        rq_set_pos_spd_for(128, 127, 127, "1")
        rq_wait_pos_spe_for_request(128, 127, 127, "1")
        rq_go_to("1")
        rq_wait("1")
        # end: URCap Program Node
        $ 793 "cur_pose≔pose_trans(pose_inv(stn5_plane), get_actual_tcp_pose())"
        global cur_pose= pose_trans ( pose_inv (stn5_plane),  get_actual_tcp_pose ())
        $ 795 "stn5_cw_pick_p≔pose_trans(cur_pose, p[0,0,stn5_pick_cw_z/1000,0,0,0])"
        global stn5_cw_pick_p= pose_trans (cur_pose, p[0,0,stn5_pick_cw_z/1000,0,0,0])
        $ 796 "FahreLinear"
        $ 797 "stn5_cw_pick_p" "breakAfter"
        set_tcp(p[-3.0E-4,2.5E-4,0.1575,0.0,0.0,0.0])
        movel(pose_trans(stn5_plane, stn5_cw_pick_p), a=0.3, v=0.1)
        # begin: URCap Program Node
        #   Source: Robotiq_Grippers, 1.8.13.22852, Robotiq Inc.
        #   Type: Greifer
        $ 798 "Greifer geschlossen (1)"
        if not(gripper_connected[0]):
          popup("Greifer 1 muss verbunden sein, um dieses Programm auszuführen.", "Keine Verbindung", False, True, True)
        end
        if not(rq_is_gripper_activated("1")):
          popup("Greifer 1 ist nicht aktiviert. Wechseln Sie zur Registerkarte Installation > Greifer, um ihn zu aktivieren und das Programm erneut auszuführen.", "Nicht aktiviert", False, True, True)
        end
        rq_set_pos_spd_for(255, 128, 128, "1")
        rq_wait_pos_spe_for_request(255, 128, 128, "1")
        rq_go_to("1")
        rq_wait("1")
        # end: URCap Program Node
        $ 799 "source_p" "breakAfter"
        set_tcp(p[-3.0E-4,2.5E-4,0.1575,0.0,0.0,0.0])
        movel(pose_trans(stn5_plane, source_p), a=0.3, v=0.1)
        $ 800 "FahreAchse"
        $ 801 "dest_p" "breakAfter"
        set_tcp(p[-3.0E-4,2.5E-4,0.1575,0.0,0.0,0.0])
        movej(pose_trans(stn5_plane, dest_p), a=1.3962634015954636, v=1.0471975511965976)
        $ 802 "cur_pose≔pose_trans(pose_inv(stn5_plane), get_actual_tcp_pose())"
        global cur_pose= pose_trans ( pose_inv (stn5_plane),  get_actual_tcp_pose ())
        $ 804 "stn5_cw_place_p≔pose_trans(cur_pose, p[0,0,stn5_place_tb_z/1000,0,0,0])"
        global stn5_cw_place_p= pose_trans (cur_pose, p[0,0,stn5_place_tb_z/1000,0,0,0])
        $ 805 "FahreLinear"
        $ 806 "stn5_cw_place_p" "breakAfter"
        set_tcp(p[-3.0E-4,2.5E-4,0.1575,0.0,0.0,0.0])
        movel(pose_trans(stn5_plane, stn5_cw_place_p), a=0.3, v=0.1)
        # begin: URCap Program Node
        #   Source: Robotiq_Grippers, 1.8.13.22852, Robotiq Inc.
        #   Type: Greifer
        $ 807 "Greiferbewegung50% (1)"
        if not(gripper_connected[0]):
          popup("Greifer 1 muss verbunden sein, um dieses Programm auszuführen.", "Keine Verbindung", False, True, True)
        end
        if not(rq_is_gripper_activated("1")):
          popup("Greifer 1 ist nicht aktiviert. Wechseln Sie zur Registerkarte Installation > Greifer, um ihn zu aktivieren und das Programm erneut auszuführen.", "Nicht aktiviert", False, True, True)
        end
        rq_set_pos_spd_for(127, 127, 127, "1")
        rq_wait_pos_spe_for_request(127, 127, 127, "1")
        rq_go_to("1")
        rq_wait("1")
        # end: URCap Program Node
        $ 808 "dest_p" "breakAfter"
        set_tcp(p[-3.0E-4,2.5E-4,0.1575,0.0,0.0,0.0])
        movel(pose_trans(stn5_plane, dest_p), a=0.3, v=0.1)
        # begin: URCap Program Node
        #   Source: Robotiq_Grippers, 1.8.13.22852, Robotiq Inc.
        #   Type: Greifer
        $ 809 "Greifer geschlossen (1)"
        if not(gripper_connected[0]):
          popup("Greifer 1 muss verbunden sein, um dieses Programm auszuführen.", "Keine Verbindung", False, True, True)
        end
        if not(rq_is_gripper_activated("1")):
          popup("Greifer 1 ist nicht aktiviert. Wechseln Sie zur Registerkarte Installation > Greifer, um ihn zu aktivieren und das Programm erneut auszuführen.", "Nicht aktiviert", False, True, True)
        end
        rq_set_pos_spd_for(255, 255, 0, "1")
        rq_wait_pos_spe_for_request(255, 255, 0, "1")
        rq_go_to("1")
        rq_wait("1")
        # end: URCap Program Node
        $ 810 "FahreAchse"
        $ 811 "stn5_stn4_hlp_p" "breakAfter"
        set_tcp(p[-3.0E-4,2.5E-4,0.1575,0.0,0.0,0.0])
        movej(get_inverse_kin(pose_trans(stn6_plane, pose_trans(p[.776557109756, -.878329076792, .250244777977, -.001605684562, .009314448336, 1.565629725105], stn5_stn4_hlp_p_p)), qnear=stn5_stn4_hlp_p_q), a=1.3962634015954636, v=1.0471975511965976)
        $ 812 "stn6_home_p" "breakAfter"
        set_tcp(p[-3.0E-4,2.5E-4,0.1575,0.0,0.0,0.0])
        movej(get_inverse_kin(pose_trans(stn6_plane, pose_trans(p[.776557109756, -.878329076792, .250244777977, -.001605684562, .009314448336, 1.565629725105], stn6_home_p_p)), qnear=stn6_home_p_q), a=1.3962634015954636, v=1.0471975511965976)
        $ 813 "Aufruf reset_jobs"
        reset_jobs()
      end
    elif (60 == switch_1):
      $ 814 "Case 60"
      $ 815 "If Test ≟  True "
      if (Test  ==    True  ):
        $ 816 "qMast.set_init_alarm(6)"
        qMast.set_init_alarm(6)
      else:
        $ 817 "Else" "noBreak"
        $ 818 "FahreAchse"
        $ 819 "stn6_home_p" "breakAfter"
        set_tcp(p[-3.0E-4,2.5E-4,0.1575,0.0,0.0,0.0])
        movej(get_inverse_kin(pose_trans(stn6_plane, pose_trans(p[.776557109756, -.878329076792, .250244777977, -.001605684562, .009314448336, 1.565629725105], stn6_home_p_p)), qnear=stn6_home_p_q), a=1.3962634015954636, v=1.0471975511965976, r=0.1)
        $ 820 "FahreAchse"
        $ 821 "stn6_help_p" "breakAfter"
        set_tcp(p[-3.0E-4,2.5E-4,0.1575,0.0,0.0,0.0])
        movej(get_inverse_kin(pose_trans(stn6_plane, pose_trans(p[.776557109756, -.878329076792, .250244777977, -.001605684562, .009314448336, 1.565629725105], stn6_help_p_p)), qnear=stn6_help_p_q), a=1.3962634015954636, v=1.0471975511965976)
        $ 822 "qMast.set_init_alarm(6)"
        qMast.set_init_alarm(6)
        $ 823 "FahreAchse"
        $ 824 "stn14_pl_rk_p" "breakAfter"
        set_tcp(p[-3.0E-4,2.5E-4,0.1575,0.0,0.0,0.0])
        movej(get_inverse_kin(pose_trans(stn6_plane, pose_trans(p[.776557109756, -.878329076792, .250244777977, -.001605684562, .009314448336, 1.565629725105], stn14_pl_rk_p_p)), qnear=stn14_pl_rk_p_q), a=1.3962634015954636, v=1.0471975511965976)
        # begin: URCap Program Node
        #   Source: Robotiq_Grippers, 1.8.13.22852, Robotiq Inc.
        #   Type: Greifer
        $ 825 "Greiferbewegung30% (1)"
        if not(gripper_connected[0]):
          popup("Greifer 1 muss verbunden sein, um dieses Programm auszuführen.", "Keine Verbindung", False, True, True)
        end
        if not(rq_is_gripper_activated("1")):
          popup("Greifer 1 ist nicht aktiviert. Wechseln Sie zur Registerkarte Installation > Greifer, um ihn zu aktivieren und das Programm erneut auszuführen.", "Nicht aktiviert", False, True, True)
        end
        rq_set_pos_spd_for(77, 255, 255, "1")
        rq_wait_pos_spe_for_request(77, 255, 255, "1")
        rq_go_to("1")
        rq_wait("1")
        # end: URCap Program Node
        $ 826 "FahreLinear"
        $ 827 "stn14_ch_rk_p" "breakAfter"
        set_tcp(p[-3.0E-4,2.5E-4,0.1575,0.0,0.0,0.0])
        movel(pose_trans(stn6_plane, pose_trans(p[.776557109756, -.878329076792, .250244777977, -.001605684562, .009314448336, 1.565629725105], stn14_ch_rk_p_p)), a=1.2, v=0.25)
        # begin: URCap Program Node
        #   Source: Robotiq_Grippers, 1.8.13.22852, Robotiq Inc.
        #   Type: Greifer
        $ 828 "Greifer geschlossen (1)"
        if not(gripper_connected[0]):
          popup("Greifer 1 muss verbunden sein, um dieses Programm auszuführen.", "Keine Verbindung", False, True, True)
        end
        if not(rq_is_gripper_activated("1")):
          popup("Greifer 1 ist nicht aktiviert. Wechseln Sie zur Registerkarte Installation > Greifer, um ihn zu aktivieren und das Programm erneut auszuführen.", "Nicht aktiviert", False, True, True)
        end
        rq_set_pos_spd_for(255, 128, 0, "1")
        rq_wait_pos_spe_for_request(255, 128, 0, "1")
        rq_go_to("1")
        rq_wait("1")
        # end: URCap Program Node
        # begin: URCap Program Node
        #   Source: Robotiq_Grippers, 1.8.13.22852, Robotiq Inc.
        #   Type: Griffkontrolle
        $ 829 "Griffkontrolle"
        # begin: URCap Program Node
        #   Source: Robotiq_Grippers, 1.8.13.22852, Robotiq Inc.
        #   Type: Wenn
        $ 830 "Wenn Objekt erkannt          " "noBreak"
        if (rq_is_object_detected(1)):
          $ 831 "qMast.stn14_fill_holder()" "noBreak"
          qMast.stn14_fill_holder()
          # end: URCap Program Node
        end
        # end: URCap Program Node
        # begin: URCap Program Node
        #   Source: Robotiq_Grippers, 1.8.13.22852, Robotiq Inc.
        #   Type: Greifer
        $ 832 "Greiferbewegung30% (1)"
        if not(gripper_connected[0]):
          popup("Greifer 1 muss verbunden sein, um dieses Programm auszuführen.", "Keine Verbindung", False, True, True)
        end
        if not(rq_is_gripper_activated("1")):
          popup("Greifer 1 ist nicht aktiviert. Wechseln Sie zur Registerkarte Installation > Greifer, um ihn zu aktivieren und das Programm erneut auszuführen.", "Nicht aktiviert", False, True, True)
        end
        rq_set_pos_spd_for(77, 255, 0, "1")
        rq_wait_pos_spe_for_request(77, 255, 0, "1")
        rq_go_to("1")
        rq_wait("1")
        # end: URCap Program Node
        $ 833 "stn14_pl_rk_p" "breakAfter"
        set_tcp(p[-3.0E-4,2.5E-4,0.1575,0.0,0.0,0.0])
        movel(pose_trans(stn6_plane, pose_trans(p[.776557109756, -.878329076792, .250244777977, -.001605684562, .009314448336, 1.565629725105], stn14_pl_rk_p_p)), a=1.2, v=0.25)
        # begin: URCap Program Node
        #   Source: Robotiq_Grippers, 1.8.13.22852, Robotiq Inc.
        #   Type: Greifer
        $ 834 "Greifer geschlossen (1)"
        if not(gripper_connected[0]):
          popup("Greifer 1 muss verbunden sein, um dieses Programm auszuführen.", "Keine Verbindung", False, True, True)
        end
        if not(rq_is_gripper_activated("1")):
          popup("Greifer 1 ist nicht aktiviert. Wechseln Sie zur Registerkarte Installation > Greifer, um ihn zu aktivieren und das Programm erneut auszuführen.", "Nicht aktiviert", False, True, True)
        end
        rq_set_pos_spd_for(255, 128, 0, "1")
        rq_wait_pos_spe_for_request(255, 128, 0, "1")
        rq_go_to("1")
        rq_wait("1")
        # end: URCap Program Node
        $ 835 "FahreAchse"
        $ 836 "stn5_chkrk_h1_p" "breakAfter"
        set_tcp(p[-3.0E-4,2.5E-4,0.1575,0.0,0.0,0.0])
        movej(get_inverse_kin(pose_trans(stn5_plane, pose_trans(p[.404793763265, -.880564591570, .218599261998, -.002768907827, .001807604230, 1.568627611983], stn5_chkrk_h1_p_p)), qnear=stn5_chkrk_h1_p_q), a=1.3962634015954636, v=1.0471975511965976)
        # begin: URCap Program Node
        #   Source: Robotiq_Grippers, 1.8.13.22852, Robotiq Inc.
        #   Type: Greifer
        $ 837 "Greifer offen (1)"
        if not(gripper_connected[0]):
          popup("Greifer 1 muss verbunden sein, um dieses Programm auszuführen.", "Keine Verbindung", False, True, True)
        end
        if not(rq_is_gripper_activated("1")):
          popup("Greifer 1 ist nicht aktiviert. Wechseln Sie zur Registerkarte Installation > Greifer, um ihn zu aktivieren und das Programm erneut auszuführen.", "Nicht aktiviert", False, True, True)
        end
        rq_set_pos_spd_for(0, 255, 127, "1")
        rq_wait_pos_spe_for_request(0, 255, 127, "1")
        rq_go_to("1")
        rq_wait("1")
        # end: URCap Program Node
        $ 838 "FahreLinear"
        $ 839 "stn5_chk_rk_1_p" "breakAfter"
        set_tcp(p[-3.0E-4,2.5E-4,0.1575,0.0,0.0,0.0])
        movel(pose_trans(stn5_plane, pose_trans(p[.404793763265, -.880564591570, .218599261998, -.002768907827, .001807604230, 1.568627611983], stn5_chk_rk_1_p_p)), a=1.0, v=0.2)
        $ 840 "Aufruf stn5_rack_check"
        stn5_rack_check()
        $ 841 "stn5_chk_rk_1_p" "breakAfter"
        set_tcp(p[-3.0E-4,2.5E-4,0.1575,0.0,0.0,0.0])
        movel(pose_trans(stn5_plane, pose_trans(p[.404793763265, -.880564591570, .218599261998, -.002768907827, .001807604230, 1.568627611983], stn5_chk_rk_1_p_p)), a=1.0, v=0.2)
        $ 842 "stn5_chk_rk_2_p" "breakAfter"
        set_tcp(p[-3.0E-4,2.5E-4,0.1575,0.0,0.0,0.0])
        movel(pose_trans(stn5_plane, pose_trans(p[.404793763265, -.880564591570, .218599261998, -.002768907827, .001807604230, 1.568627611983], stn5_chk_rk_2_p_p)), a=1.0, v=0.2)
        $ 843 "Aufruf stn5_rack_check"
        stn5_rack_check()
        $ 844 "stn5_chk_rk_2_p" "breakAfter"
        set_tcp(p[-3.0E-4,2.5E-4,0.1575,0.0,0.0,0.0])
        movel(pose_trans(stn5_plane, pose_trans(p[.404793763265, -.880564591570, .218599261998, -.002768907827, .001807604230, 1.568627611983], stn5_chk_rk_2_p_p)), a=1.0, v=0.2)
        $ 845 "stn5_chk_rk_3_p" "breakAfter"
        set_tcp(p[-3.0E-4,2.5E-4,0.1575,0.0,0.0,0.0])
        movel(pose_trans(stn5_plane, pose_trans(p[.404793763265, -.880564591570, .218599261998, -.002768907827, .001807604230, 1.568627611983], stn5_chk_rk_3_p_p)), a=1.0, v=0.2)
        $ 846 "Aufruf stn5_rack_check"
        stn5_rack_check()
        $ 847 "stn5_chk_rk_3_p" "breakAfter"
        set_tcp(p[-3.0E-4,2.5E-4,0.1575,0.0,0.0,0.0])
        movel(pose_trans(stn5_plane, pose_trans(p[.404793763265, -.880564591570, .218599261998, -.002768907827, .001807604230, 1.568627611983], stn5_chk_rk_3_p_p)), a=1.0, v=0.2)
        $ 848 "stn5_chk_rk_4_p" "breakAfter"
        set_tcp(p[-3.0E-4,2.5E-4,0.1575,0.0,0.0,0.0])
        movel(pose_trans(stn5_plane, pose_trans(p[.404793763265, -.880564591570, .218599261998, -.002768907827, .001807604230, 1.568627611983], stn5_chk_rk_4_p_p)), a=1.0, v=0.2)
        $ 849 "Aufruf stn5_rack_check"
        stn5_rack_check()
        $ 850 "stn5_chk_rk_4_p" "breakAfter"
        set_tcp(p[-3.0E-4,2.5E-4,0.1575,0.0,0.0,0.0])
        movel(pose_trans(stn5_plane, pose_trans(p[.404793763265, -.880564591570, .218599261998, -.002768907827, .001807604230, 1.568627611983], stn5_chk_rk_4_p_p)), a=1.0, v=0.2)
        $ 851 "stn5_chkrk_h2_p" "breakAfter"
        set_tcp(p[-3.0E-4,2.5E-4,0.1575,0.0,0.0,0.0])
        movel(pose_trans(stn5_plane, pose_trans(p[.404793763265, -.880564591570, .218599261998, -.002768907827, .001807604230, 1.568627611983], stn5_chkrk_h2_p_p)), a=1.0, v=0.2)
        $ 852 "stn5_chkrk_h3_p" "breakAfter"
        set_tcp(p[-3.0E-4,2.5E-4,0.1575,0.0,0.0,0.0])
        movel(pose_trans(stn5_plane, pose_trans(p[.404793763265, -.880564591570, .218599261998, -.002768907827, .001807604230, 1.568627611983], stn5_chkrk_h3_p_p)), a=1.0, v=0.2)
        $ 853 "stn5_chk_rk_5_p" "breakAfter"
        set_tcp(p[-3.0E-4,2.5E-4,0.1575,0.0,0.0,0.0])
        movel(pose_trans(stn5_plane, pose_trans(p[.404793763265, -.880564591570, .218599261998, -.002768907827, .001807604230, 1.568627611983], stn5_chk_rk_5_p_p)), a=1.0, v=0.2)
        $ 854 "Aufruf stn5_rack_check"
        stn5_rack_check()
        $ 855 "stn5_chk_rk_5_p" "breakAfter"
        set_tcp(p[-3.0E-4,2.5E-4,0.1575,0.0,0.0,0.0])
        movel(pose_trans(stn5_plane, pose_trans(p[.404793763265, -.880564591570, .218599261998, -.002768907827, .001807604230, 1.568627611983], stn5_chk_rk_5_p_p)), a=1.0, v=0.2)
        $ 856 "stn5_chk_rk_6_p" "breakAfter"
        set_tcp(p[-3.0E-4,2.5E-4,0.1575,0.0,0.0,0.0])
        movel(pose_trans(stn5_plane, pose_trans(p[.404793763265, -.880564591570, .218599261998, -.002768907827, .001807604230, 1.568627611983], stn5_chk_rk_6_p_p)), a=1.0, v=0.2)
        $ 857 "Aufruf stn5_rack_check"
        stn5_rack_check()
        $ 858 "stn5_chk_rk_6_p" "breakAfter"
        set_tcp(p[-3.0E-4,2.5E-4,0.1575,0.0,0.0,0.0])
        movel(pose_trans(stn5_plane, pose_trans(p[.404793763265, -.880564591570, .218599261998, -.002768907827, .001807604230, 1.568627611983], stn5_chk_rk_6_p_p)), a=1.0, v=0.2)
        $ 859 "stn5_chk_rk_7_p" "breakAfter"
        set_tcp(p[-3.0E-4,2.5E-4,0.1575,0.0,0.0,0.0])
        movel(pose_trans(stn5_plane, pose_trans(p[.404793763265, -.880564591570, .218599261998, -.002768907827, .001807604230, 1.568627611983], stn5_chk_rk_7_p_p)), a=1.0, v=0.2)
        $ 860 "Aufruf stn5_rack_check"
        stn5_rack_check()
        $ 861 "stn5_chk_rk_7_p" "breakAfter"
        set_tcp(p[-3.0E-4,2.5E-4,0.1575,0.0,0.0,0.0])
        movel(pose_trans(stn5_plane, pose_trans(p[.404793763265, -.880564591570, .218599261998, -.002768907827, .001807604230, 1.568627611983], stn5_chk_rk_7_p_p)), a=1.0, v=0.2)
        $ 862 "stn5_chk_rk_8_p" "breakAfter"
        set_tcp(p[-3.0E-4,2.5E-4,0.1575,0.0,0.0,0.0])
        movel(pose_trans(stn5_plane, pose_trans(p[.404793763265, -.880564591570, .218599261998, -.002768907827, .001807604230, 1.568627611983], stn5_chk_rk_8_p_p)), a=1.0, v=0.2)
        $ 863 "Aufruf stn5_rack_check"
        stn5_rack_check()
        $ 864 "stn5_chk_rk_8_p" "breakAfter"
        set_tcp(p[-3.0E-4,2.5E-4,0.1575,0.0,0.0,0.0])
        movel(pose_trans(stn5_plane, pose_trans(p[.404793763265, -.880564591570, .218599261998, -.002768907827, .001807604230, 1.568627611983], stn5_chk_rk_8_p_p)), a=1.0, v=0.2)
        $ 865 "stn5_chkrk_h4_p" "breakAfter"
        set_tcp(p[-3.0E-4,2.5E-4,0.1575,0.0,0.0,0.0])
        movel(pose_trans(stn5_plane, pose_trans(p[.404793763265, -.880564591570, .218599261998, -.002768907827, .001807604230, 1.568627611983], stn5_chkrk_h4_p_p)), a=1.0, v=0.2)
        # begin: URCap Program Node
        #   Source: Robotiq_Grippers, 1.8.13.22852, Robotiq Inc.
        #   Type: Greifer
        $ 866 "Greifer geschlossen (1)"
        if not(gripper_connected[0]):
          popup("Greifer 1 muss verbunden sein, um dieses Programm auszuführen.", "Keine Verbindung", False, True, True)
        end
        if not(rq_is_gripper_activated("1")):
          popup("Greifer 1 ist nicht aktiviert. Wechseln Sie zur Registerkarte Installation > Greifer, um ihn zu aktivieren und das Programm erneut auszuführen.", "Nicht aktiviert", False, True, True)
        end
        rq_set_pos_spd_for(255, 255, 127, "1")
        rq_wait_pos_spe_for_request(255, 255, 127, "1")
        rq_go_to("1")
        rq_wait("1")
        # end: URCap Program Node
        $ 867 "FahreAchse"
        $ 868 "stn6_home_p" "breakAfter"
        set_tcp(p[-3.0E-4,2.5E-4,0.1575,0.0,0.0,0.0])
        movej(get_inverse_kin(pose_trans(stn6_plane, pose_trans(p[.776557109756, -.878329076792, .250244777977, -.001605684562, .009314448336, 1.565629725105], stn6_home_p_p)), qnear=stn6_home_p_q), a=1.3962634015954636, v=1.0471975511965976)
        $ 869 "If archiv_opened ≟  False "
        if (archiv_opened  ==    False  ):
          $ 870 "Aufruf stn11_open_archiv"
          stn11_open_archiv()
          $ 871 "archiv_opened≔ True "
          global archiv_opened=  True
        end
        $ 872 "FahreAchse"
        $ 873 "stn6_home_p" "breakAfter"
        set_tcp(p[-3.0E-4,2.5E-4,0.1575,0.0,0.0,0.0])
        movej(get_inverse_kin(pose_trans(stn6_plane, pose_trans(p[.776557109756, -.878329076792, .250244777977, -.001605684562, .009314448336, 1.565629725105], stn6_home_p_p)), qnear=stn6_home_p_q), a=1.3962634015954636, v=1.0471975511965976)
      end
      $ 874 "Aufruf reset_jobs"
      reset_jobs()
    elif (61 == switch_1):
      $ 875 "Case 61"
      $ 876 "FahreAchse"
      $ 877 "stn6_home_p" "breakAfter"
      set_tcp(p[-3.0E-4,2.5E-4,0.1575,0.0,0.0,0.0])
      movej(get_inverse_kin(pose_trans(stn6_plane, pose_trans(p[.776557109756, -.878329076792, .250244777977, -.001605684562, .009314448336, 1.565629725105], stn6_home_p_p)), qnear=stn6_home_p_q), a=1.3962634015954636, v=1.0471975511965976, r=0.1)
      $ 878 "stn6_help_p" "breakAfter"
      set_tcp(p[-3.0E-4,2.5E-4,0.1575,0.0,0.0,0.0])
      movej(get_inverse_kin(pose_trans(stn6_plane, pose_trans(p[.776557109756, -.878329076792, .250244777977, -.001605684562, .009314448336, 1.565629725105], stn6_help_p_p)), qnear=stn6_help_p_q), a=1.3962634015954636, v=1.0471975511965976)
      $ 879 "dest_jobID≔jobArr[1]"
      global dest_jobID=jobArr[1]
      $ 880 "stn5_dest_4ps_p≔qMast.stn5_get_loc()"
      global stn5_dest_4ps_p=qMast.stn5_get_loc()
      $ 881 "If Test ≟  True "
      if (Test  ==    True  ):
        $ 882 "Kommentar"
        # Kommentar
      else:
        $ 883 "Else" "noBreak"
        $ 884 "stn6_hatch_open≔qMast.stn6_hatch_open()"
        global stn6_hatch_open=qMast.stn6_hatch_open()
        $ 885 "If stn6_hatch_open ≟  True "
        if (stn6_hatch_open  ==    True  ):
          $ 886 "stn5_loop_count≔0"
          global stn5_loop_count=0
          $ 887 "Schleife 4 mal"
          Loop_1 = 0
          while (Loop_1 < 4):
            $ 888 "FahreAchse"
            $ 889 "stn6_help_p" "breakAfter"
            set_tcp(p[-3.0E-4,2.5E-4,0.1575,0.0,0.0,0.0])
            movej(get_inverse_kin(pose_trans(stn6_plane, pose_trans(p[.776557109756, -.878329076792, .250244777977, -.001605684562, .009314448336, 1.565629725105], stn6_help_p_p)), qnear=stn6_help_p_q), a=1.3962634015954636, v=1.0471975511965976)
            $ 890 "stn6_set_rotor≔qMast.stn6_set_rotor_position(stn5_loop_count + 1)"
            global stn6_set_rotor=qMast.stn6_set_rotor_position(stn5_loop_count + 1)
            $ 891 "If stn6_set_rotor ≟  True "
            if (stn6_set_rotor  ==    True  ):
              $ 892 "FahreAchse"
              $ 893 "stn6_place_p" "breakAfter"
              set_tcp(p[-3.0E-4,2.5E-4,0.1575,0.0,0.0,0.0])
              movej(get_inverse_kin(pose_trans(stn6_plane, pose_trans(p[.776557109756, -.878329076792, .250244777977, -.001605684562, .009314448336, 1.565629725105], stn6_place_p_p)), qnear=stn6_place_p_q), a=1.3962634015954636, v=1.0471975511965976)
              # begin: URCap Program Node
              #   Source: Robotiq_Grippers, 1.8.13.22852, Robotiq Inc.
              #   Type: Greifer
              $ 894 "Greiferbewegung40% (1)"
              if not(gripper_connected[0]):
                popup("Greifer 1 muss verbunden sein, um dieses Programm auszuführen.", "Keine Verbindung", False, True, True)
              end
              if not(rq_is_gripper_activated("1")):
                popup("Greifer 1 ist nicht aktiviert. Wechseln Sie zur Registerkarte Installation > Greifer, um ihn zu aktivieren und das Programm erneut auszuführen.", "Nicht aktiviert", False, True, True)
              end
              rq_set_pos_spd_for(102, 255, 0, "1")
              rq_wait_pos_spe_for_request(102, 255, 0, "1")
              rq_go_to("1")
              rq_wait("1")
              # end: URCap Program Node
              $ 895 "FahreLinear"
              $ 896 "cur_pose≔pose_trans(pose_inv(stn6_plane), get_actual_tcp_pose())"
              global cur_pose= pose_trans ( pose_inv (stn6_plane),  get_actual_tcp_pose ())
              $ 898 "stn6_pick_z_p≔pose_trans(cur_pose, p[0,0,stn6_pick_z/1000,0,0,0])"
              global stn6_pick_z_p= pose_trans (cur_pose, p[0,0,stn6_pick_z/1000,0,0,0])
              $ 899 "stn6_pick_z_p" "breakAfter"
              set_tcp(p[-3.0E-4,2.5E-4,0.1575,0.0,0.0,0.0])
              movel(pose_trans(stn6_plane, stn6_pick_z_p), a=1.2, v=0.25)
              # begin: URCap Program Node
              #   Source: Robotiq_Grippers, 1.8.13.22852, Robotiq Inc.
              #   Type: Greifer
              $ 900 "Greifer geschlossen (1)"
              if not(gripper_connected[0]):
                popup("Greifer 1 muss verbunden sein, um dieses Programm auszuführen.", "Keine Verbindung", False, True, True)
              end
              if not(rq_is_gripper_activated("1")):
                popup("Greifer 1 ist nicht aktiviert. Wechseln Sie zur Registerkarte Installation > Greifer, um ihn zu aktivieren und das Programm erneut auszuführen.", "Nicht aktiviert", False, True, True)
              end
              rq_set_pos_spd_for(255, 128, 128, "1")
              rq_wait_pos_spe_for_request(255, 128, 128, "1")
              rq_go_to("1")
              rq_wait("1")
              # end: URCap Program Node
              $ 901 "stn6_place_p" "breakAfter"
              set_tcp(p[-3.0E-4,2.5E-4,0.1575,0.0,0.0,0.0])
              movel(pose_trans(stn6_plane, pose_trans(p[.776557109756, -.878329076792, .250244777977, -.001605684562, .009314448336, 1.565629725105], stn6_place_p_p)), a=1.2, v=0.25)
              $ 902 "stn5_source_p≔stn5_dest_4ps_p[stn5_loop_count]"
              global stn5_source_p=stn5_dest_4ps_p[stn5_loop_count]
              $ 903 "FahreAchse"
              $ 904 "stn6_help_p" "breakAfter"
              set_tcp(p[-3.0E-4,2.5E-4,0.1575,0.0,0.0,0.0])
              movej(get_inverse_kin(pose_trans(stn6_plane, pose_trans(p[.776557109756, -.878329076792, .250244777977, -.001605684562, .009314448336, 1.565629725105], stn6_help_p_p)), qnear=stn6_help_p_q), a=1.3962634015954636, v=1.0471975511965976, r=0.05)
              $ 905 "FahreAchse"
              $ 906 "stn5_source_p" "breakAfter"
              set_tcp(p[-3.0E-4,2.5E-4,0.1575,0.0,0.0,0.0])
              movej(pose_trans(stn5_plane, stn5_source_p), a=1.3962634015954636, v=1.0471975511965976)
              $ 907 "FahreLinear"
              $ 908 "cur_pose≔pose_trans(pose_inv(stn5_plane), get_actual_tcp_pose())"
              global cur_pose= pose_trans ( pose_inv (stn5_plane),  get_actual_tcp_pose ())
              $ 909 "stn5_place_rk_p≔pose_trans(cur_pose, p[0,0,stn5_place_rk_z/1000,0,0,0])"
              global stn5_place_rk_p= pose_trans (cur_pose, p[0,0,stn5_place_rk_z/1000,0,0,0])
              $ 910 "stn5_place_rk_p" "breakAfter"
              set_tcp(p[-3.0E-4,2.5E-4,0.1575,0.0,0.0,0.0])
              movel(pose_trans(stn5_plane, stn5_place_rk_p), a=0.6, v=0.1)
              # begin: URCap Program Node
              #   Source: Robotiq_Grippers, 1.8.13.22852, Robotiq Inc.
              #   Type: Greifer
              $ 911 "Greiferbewegung50% (1)"
              if not(gripper_connected[0]):
                popup("Greifer 1 muss verbunden sein, um dieses Programm auszuführen.", "Keine Verbindung", False, True, True)
              end
              if not(rq_is_gripper_activated("1")):
                popup("Greifer 1 ist nicht aktiviert. Wechseln Sie zur Registerkarte Installation > Greifer, um ihn zu aktivieren und das Programm erneut auszuführen.", "Nicht aktiviert", False, True, True)
              end
              rq_set_pos_spd_for(128, 255, 255, "1")
              rq_wait_pos_spe_for_request(128, 255, 255, "1")
              rq_go_to("1")
              rq_wait("1")
              # end: URCap Program Node
              $ 912 "stn5_source_p" "breakAfter"
              set_tcp(p[-3.0E-4,2.5E-4,0.1575,0.0,0.0,0.0])
              movel(pose_trans(stn5_plane, stn5_source_p), a=1.2, v=0.25)
              # begin: URCap Program Node
              #   Source: Robotiq_Grippers, 1.8.13.22852, Robotiq Inc.
              #   Type: Greifer
              $ 913 "Greifer geschlossen (1)"
              if not(gripper_connected[0]):
                popup("Greifer 1 muss verbunden sein, um dieses Programm auszuführen.", "Keine Verbindung", False, True, True)
              end
              if not(rq_is_gripper_activated("1")):
                popup("Greifer 1 ist nicht aktiviert. Wechseln Sie zur Registerkarte Installation > Greifer, um ihn zu aktivieren und das Programm erneut auszuführen.", "Nicht aktiviert", False, True, True)
              end
              rq_set_pos_spd_for(255, 255, 255, "1")
              rq_wait_pos_spe_for_request(255, 255, 255, "1")
              rq_go_to("1")
              rq_wait("1")
              # end: URCap Program Node
              $ 914 "stn5_loop_count≔stn5_loop_count + 1"
              global stn5_loop_count=stn5_loop_count + 1
            end
            Loop_1 = Loop_1 + 1
          end
        end
      end
      $ 915 "FahreAchse"
      $ 916 "stn6_help_p" "breakAfter"
      set_tcp(p[-3.0E-4,2.5E-4,0.1575,0.0,0.0,0.0])
      movej(get_inverse_kin(pose_trans(stn6_plane, pose_trans(p[.776557109756, -.878329076792, .250244777977, -.001605684562, .009314448336, 1.565629725105], stn6_help_p_p)), qnear=stn6_help_p_q), a=1.3962634015954636, v=1.0471975511965976)
      $ 917 "stn6_home_p" "breakAfter"
      set_tcp(p[-3.0E-4,2.5E-4,0.1575,0.0,0.0,0.0])
      movej(get_inverse_kin(pose_trans(stn6_plane, pose_trans(p[.776557109756, -.878329076792, .250244777977, -.001605684562, .009314448336, 1.565629725105], stn6_home_p_p)), qnear=stn6_home_p_q), a=1.3962634015954636, v=1.0471975511965976)
      $ 918 "Aufruf reset_jobs"
      reset_jobs()
    elif (70 == switch_1):
      $ 919 "Case 70"
      $ 920 "If Test ≟  True "
      if (Test  ==    True  ):
        $ 921 "qMast.set_init_alarm(7)"
        qMast.set_init_alarm(7)
      else:
        $ 922 "Else" "noBreak"
        $ 923 "Aufruf stn7_close_doors"
        stn7_close_doors()
        $ 924 "Aufruf stn7_init_stndby"
        stn7_init_stndby()
        $ 925 "If archiv_opened ≟  False "
        if (archiv_opened  ==    False  ):
          $ 926 "Aufruf stn11_open_archiv"
          stn11_open_archiv()
          $ 927 "archiv_opened≔ True "
          global archiv_opened=  True
        end
      end
      $ 928 "Aufruf reset_jobs"
      reset_jobs()
    elif (71 == switch_1):
      $ 929 "Case 71"
      $ 930 "FahreAchse"
      $ 931 "stn7_home_p" "breakAfter"
      set_tcp(p[-3.0E-4,2.5E-4,0.1575,0.0,0.0,0.0])
      movej(get_inverse_kin(pose_trans(stn7_plane, pose_trans(p[.109811488584, -1.023382701287, -.166619380160, .003048702642, -.008599620441, 2.442192581404], stn7_home_p_p)), qnear=stn7_home_p_q), a=1.3962634015954636, v=1.0471975511965976, r=0.1)
      $ 932 "src_dest_p≔qMast.get_loc()"
      global src_dest_p=qMast.get_loc()
      $ 933 "source_p≔src_dest_p[0]"
      global source_p=src_dest_p[0]
      $ 934 "FahreAchse"
      $ 935 "source_p" "breakAfter"
      set_tcp(p[-3.0E-4,2.5E-4,0.1575,0.0,0.0,0.0])
      movej(pose_trans(stn7_plane, source_p), a=1.3962634015954636, v=1.0471975511965976)
      $ 936 "FahreLinear"
      # begin: URCap Program Node
      #   Source: Robotiq_Grippers, 1.8.13.22852, Robotiq Inc.
      #   Type: Greifer
      $ 937 "Greifer offen (1)"
      if not(gripper_connected[0]):
        popup("Greifer 1 muss verbunden sein, um dieses Programm auszuführen.", "Keine Verbindung", False, True, True)
      end
      if not(rq_is_gripper_activated("1")):
        popup("Greifer 1 ist nicht aktiviert. Wechseln Sie zur Registerkarte Installation > Greifer, um ihn zu aktivieren und das Programm erneut auszuführen.", "Nicht aktiviert", False, True, True)
      end
      rq_set_pos_spd_for(0, 255, 0, "1")
      rq_wait_pos_spe_for_request(0, 255, 0, "1")
      rq_go_to("1")
      rq_wait("1")
      # end: URCap Program Node
      $ 938 "cur_pose≔pose_trans(pose_inv(stn7_plane), get_actual_tcp_pose())"
      global cur_pose= pose_trans ( pose_inv (stn7_plane),  get_actual_tcp_pose ())
      $ 940 "stn7_pick_z_p≔pose_trans(cur_pose, p[0,0,stn7_pick_z/1000,0,0,0])"
      global stn7_pick_z_p= pose_trans (cur_pose, p[0,0,stn7_pick_z/1000,0,0,0])
      $ 941 "stn7_pick_z_p" "breakAfter"
      set_tcp(p[-3.0E-4,2.5E-4,0.1575,0.0,0.0,0.0])
      movel(pose_trans(stn7_plane, stn7_pick_z_p), a=1.2, v=0.25)
      # begin: URCap Program Node
      #   Source: Robotiq_Grippers, 1.8.13.22852, Robotiq Inc.
      #   Type: Greifer
      $ 942 "Greifer geschlossen (1)"
      if not(gripper_connected[0]):
        popup("Greifer 1 muss verbunden sein, um dieses Programm auszuführen.", "Keine Verbindung", False, True, True)
      end
      if not(rq_is_gripper_activated("1")):
        popup("Greifer 1 ist nicht aktiviert. Wechseln Sie zur Registerkarte Installation > Greifer, um ihn zu aktivieren und das Programm erneut auszuführen.", "Nicht aktiviert", False, True, True)
      end
      rq_set_pos_spd_for(255, 128, 255, "1")
      rq_wait_pos_spe_for_request(255, 128, 255, "1")
      rq_go_to("1")
      rq_wait("1")
      # end: URCap Program Node
      $ 943 "source_p" "breakAfter"
      set_tcp(p[-3.0E-4,2.5E-4,0.1575,0.0,0.0,0.0])
      movel(pose_trans(stn7_plane, source_p), a=1.2, v=0.25)
      $ 944 "FahreLinear"
      $ 945 "stn7_bin_help_p" "breakAfter"
      set_tcp(p[-3.0E-4,2.5E-4,0.1575,0.0,0.0,0.0])
      movel(pose_trans(stn7_plane, pose_trans(p[.109811488584, -1.023382701287, -.166619380160, .003048702642, -.008599620441, 2.442192581404], stn7_bin_help_p_p)), a=1.2, v=0.6, r=0.025)
      $ 946 "FahreAchse"
      $ 947 "stn7_bin_apr_p" "breakAfter"
      set_tcp(p[-3.0E-4,2.5E-4,0.1575,0.0,0.0,0.0])
      movej(get_inverse_kin(pose_trans(stn7_plane, pose_trans(p[.109811488584, -1.023382701287, -.166619380160, .003048702642, -.008599620441, 2.442192581404], stn7_bin_apr_p_p)), qnear=stn7_bin_apr_p_q), a=1.7453292519943295, v=1.3962634015954636, r=0.02)
      $ 948 "stn7_bin_thrw_p" "breakAfter"
      set_tcp(p[-3.0E-4,2.5E-4,0.1575,0.0,0.0,0.0])
      movej(get_inverse_kin(pose_trans(stn7_plane, pose_trans(p[.109811488584, -1.023382701287, -.166619380160, .003048702642, -.008599620441, 2.442192581404], stn7_bin_thrw_p_p)), qnear=stn7_bin_thrw_p_q), a=1.3962634015954636, v=1.0471975511965976)
      # begin: URCap Program Node
      #   Source: Robotiq_Grippers, 1.8.13.22852, Robotiq Inc.
      #   Type: Greifer
      $ 949 "Greifer offen (1)"
      if not(gripper_connected[0]):
        popup("Greifer 1 muss verbunden sein, um dieses Programm auszuführen.", "Keine Verbindung", False, True, True)
      end
      if not(rq_is_gripper_activated("1")):
        popup("Greifer 1 ist nicht aktiviert. Wechseln Sie zur Registerkarte Installation > Greifer, um ihn zu aktivieren und das Programm erneut auszuführen.", "Nicht aktiviert", False, True, True)
      end
      rq_set_pos_spd_for(0, 255, 255, "1")
      rq_wait_pos_spe_for_request(0, 255, 255, "1")
      rq_go_to("1")
      rq_wait("1")
      # end: URCap Program Node
      $ 950 "Warten: 0.1"
      sleep(0.1)
      $ 951 "stn7_bin_apr_p" "breakAfter"
      set_tcp(p[-3.0E-4,2.5E-4,0.1575,0.0,0.0,0.0])
      movej(get_inverse_kin(pose_trans(stn7_plane, pose_trans(p[.109811488584, -1.023382701287, -.166619380160, .003048702642, -.008599620441, 2.442192581404], stn7_bin_apr_p_p)), qnear=stn7_bin_apr_p_q), a=1.7453292519943295, v=1.3962634015954636)
      # begin: URCap Program Node
      #   Source: Robotiq_Grippers, 1.8.13.22852, Robotiq Inc.
      #   Type: Greifer
      $ 952 "Greifer geschlossen (1)"
      if not(gripper_connected[0]):
        popup("Greifer 1 muss verbunden sein, um dieses Programm auszuführen.", "Keine Verbindung", False, True, True)
      end
      if not(rq_is_gripper_activated("1")):
        popup("Greifer 1 ist nicht aktiviert. Wechseln Sie zur Registerkarte Installation > Greifer, um ihn zu aktivieren und das Programm erneut auszuführen.", "Nicht aktiviert", False, True, True)
      end
      rq_set_pos_spd_for(255, 128, 255, "1")
      rq_wait_pos_spe_for_request(255, 128, 255, "1")
      rq_go_to("1")
      rq_wait("1")
      # end: URCap Program Node
      $ 953 "stn7_bin_help_p" "breakAfter"
      set_tcp(p[-3.0E-4,2.5E-4,0.1575,0.0,0.0,0.0])
      movej(get_inverse_kin(pose_trans(stn7_plane, pose_trans(p[.109811488584, -1.023382701287, -.166619380160, .003048702642, -.008599620441, 2.442192581404], stn7_bin_help_p_p)), qnear=stn7_bin_help_p_q), a=1.7453292519943295, v=1.3962634015954636, r=0.05)
      $ 954 "stn7_home_p" "breakAfter"
      set_tcp(p[-3.0E-4,2.5E-4,0.1575,0.0,0.0,0.0])
      movej(get_inverse_kin(pose_trans(stn7_plane, pose_trans(p[.109811488584, -1.023382701287, -.166619380160, .003048702642, -.008599620441, 2.442192581404], stn7_home_p_p)), qnear=stn7_home_p_q), a=1.3962634015954636, v=1.0471975511965976)
      $ 955 "Aufruf reset_jobs"
      reset_jobs()
    elif (73 == switch_1):
      $ 956 "Case 73"
      $ 957 "FahreAchse"
      $ 958 "stn7_home_p" "breakAfter"
      set_tcp(p[-3.0E-4,2.5E-4,0.1575,0.0,0.0,0.0])
      movej(get_inverse_kin(pose_trans(stn7_plane, pose_trans(p[.109811488584, -1.023382701287, -.166619380160, .003048702642, -.008599620441, 2.442192581404], stn7_home_p_p)), qnear=stn7_home_p_q), a=1.3962634015954636, v=1.0471975511965976)
      # begin: URCap Program Node
      #   Source: Robotiq_Grippers, 1.8.13.22852, Robotiq Inc.
      #   Type: Greifer
      $ 959 "Greifer geschlossen (1)"
      if not(gripper_connected[0]):
        popup("Greifer 1 muss verbunden sein, um dieses Programm auszuführen.", "Keine Verbindung", False, True, True)
      end
      if not(rq_is_gripper_activated("1")):
        popup("Greifer 1 ist nicht aktiviert. Wechseln Sie zur Registerkarte Installation > Greifer, um ihn zu aktivieren und das Programm erneut auszuführen.", "Nicht aktiviert", False, True, True)
      end
      rq_set_pos_spd_for(255, 128, 255, "1")
      rq_wait_pos_spe_for_request(255, 128, 255, "1")
      rq_go_to("1")
      rq_wait("1")
      # end: URCap Program Node
      $ 960 "stn7_ld_apr_p" "breakAfter"
      set_tcp(p[-3.0E-4,2.5E-4,0.1575,0.0,0.0,0.0])
      movej(get_inverse_kin(pose_trans(stn7_plane, pose_trans(p[.109811488584, -1.023382701287, -.166619380160, .003048702642, -.008599620441, 2.442192581404], stn7_ld_apr_p_p)), qnear=stn7_ld_apr_p_q), a=1.3962634015954636, v=1.0471975511965976)
      $ 961 "FahreLinear"
      $ 962 "stn7_ld_press_p" "breakAfter"
      set_tcp(p[-3.0E-4,2.5E-4,0.1575,0.0,0.0,0.0])
      movel(pose_trans(stn7_plane, pose_trans(p[.109811488584, -1.023382701287, -.166619380160, .003048702642, -.008599620441, 2.442192581404], stn7_ld_press_p_p)), a=0.6, v=0.1)
      $ 963 "stn7_ld_apr_p" "breakAfter"
      set_tcp(p[-3.0E-4,2.5E-4,0.1575,0.0,0.0,0.0])
      movel(pose_trans(stn7_plane, pose_trans(p[.109811488584, -1.023382701287, -.166619380160, .003048702642, -.008599620441, 2.442192581404], stn7_ld_apr_p_p)), a=0.6, v=0.1)
      $ 964 "qMast.set_runtime_alarm(7)"
      qMast.set_runtime_alarm(7)
      $ 965 "FahreAchse"
      $ 966 "stn7_home_p" "breakAfter"
      set_tcp(p[-3.0E-4,2.5E-4,0.1575,0.0,0.0,0.0])
      movej(get_inverse_kin(pose_trans(stn7_plane, pose_trans(p[.109811488584, -1.023382701287, -.166619380160, .003048702642, -.008599620441, 2.442192581404], stn7_home_p_p)), qnear=stn7_home_p_q), a=1.3962634015954636, v=1.0471975511965976)
      $ 967 "Aufruf reset_jobs"
      reset_jobs()
    elif (74 == switch_1):
      $ 968 "Case 74"
      $ 969 "Aufruf stn7_close_doors"
      stn7_close_doors()
      $ 970 "Aufruf stn7_open_doors"
      stn7_open_doors()
      $ 971 "Aufruf reset_jobs"
      reset_jobs()
    elif (75 == switch_1):
      $ 972 "Case 75"
      $ 973 "Aufruf stn7_close_doors"
      stn7_close_doors()
      $ 974 "FahreAchse"
      $ 975 "stn7_home_p" "breakAfter"
      set_tcp(p[-3.0E-4,2.5E-4,0.1575,0.0,0.0,0.0])
      movej(get_inverse_kin(pose_trans(stn7_plane, pose_trans(p[.109811488584, -1.023382701287, -.166619380160, .003048702642, -.008599620441, 2.442192581404], stn7_home_p_p)), qnear=stn7_home_p_q), a=1.3962634015954636, v=1.0471975511965976)
      $ 976 "Aufruf reset_jobs"
      reset_jobs()
    elif (103 == switch_1):
      $ 977 "Case 103"
      $ 978 "FahreAchse"
      $ 979 "stn1_home_p" "breakAfter"
      set_tcp(p[-3.0E-4,2.5E-4,0.1575,0.0,0.0,0.0])
      movej(get_inverse_kin(pose_trans(stn1_plane, pose_trans(p[.053539610991, -.984987293150, -.024848236577, .000189536594, .000276418508, 3.136265531618], stn1_home_p_p)), qnear=stn1_home_p_q), a=1.3962634015954636, v=1.0471975511965976, r=0.05)
      $ 980 "home_p" "breakAfter"
      set_tcp(p[-3.0E-4,2.5E-4,0.1575,0.0,0.0,0.0])
      movej(get_inverse_kin(pose_trans(stn1_plane, pose_trans(p[.053539610991, -.984987293150, -.024848236577, .000189536594, .000276418508, 3.136265531618], home_p_p)), qnear=home_p_q), a=1.3962634015954636, v=1.0471975511965976)
      $ 982 "Meldung"
      popup(str_cat("",stn10_skype_ful), "Fehler", False, True, blocking=False)
      halt
      $ 983 "Aufruf reset_jobs"
      reset_jobs()
    elif (113 == switch_1):
      $ 984 "Case 113"
      $ 985 "FahreAchse"
      $ 986 "stn1_home_p" "breakAfter"
      set_tcp(p[-3.0E-4,2.5E-4,0.1575,0.0,0.0,0.0])
      movej(get_inverse_kin(pose_trans(stn1_plane, pose_trans(p[.053539610991, -.984987293150, -.024848236577, .000189536594, .000276418508, 3.136265531618], stn1_home_p_p)), qnear=stn1_home_p_q), a=1.3962634015954636, v=1.0471975511965976, r=0.05)
      $ 987 "home_p" "breakAfter"
      set_tcp(p[-3.0E-4,2.5E-4,0.1575,0.0,0.0,0.0])
      movej(get_inverse_kin(pose_trans(stn1_plane, pose_trans(p[.053539610991, -.984987293150, -.024848236577, .000189536594, .000276418508, 3.136265531618], home_p_p)), qnear=home_p_q), a=1.3962634015954636, v=1.0471975511965976)
      $ 989 "Meldung"
      popup(str_cat("",stn11_skype_ful), "Fehler", False, True, blocking=False)
      halt
      $ 990 "Aufruf reset_jobs"
      reset_jobs()
    elif (141 == switch_1):
      $ 991 "Case 141"
      $ 992 "dest_jobID≔jobArr[1]"
      global dest_jobID=jobArr[1]
      $ 993 "FahreAchse"
      $ 994 "stn6_home_p" "breakAfter"
      set_tcp(p[-3.0E-4,2.5E-4,0.1575,0.0,0.0,0.0])
      movej(get_inverse_kin(pose_trans(stn6_plane, pose_trans(p[.776557109756, -.878329076792, .250244777977, -.001605684562, .009314448336, 1.565629725105], stn6_home_p_p)), qnear=stn6_home_p_q), a=1.3962634015954636, v=1.0471975511965976)
      $ 995 "stn14_pkrk_up_p" "breakAfter"
      set_tcp(p[-3.0E-4,2.5E-4,0.1575,0.0,0.0,0.0])
      movej(get_inverse_kin(pose_trans(stn6_plane, pose_trans(p[.776557109756, -.878329076792, .250244777977, -.001605684562, .009314448336, 1.565629725105], stn14_pkrk_up_p_p)), qnear=stn14_pkrk_up_p_q), a=1.3962634015954636, v=1.0471975511965976)
      # begin: URCap Program Node
      #   Source: Robotiq_Grippers, 1.8.13.22852, Robotiq Inc.
      #   Type: Greifer
      $ 996 "Greifer offen (1)"
      if not(gripper_connected[0]):
        popup("Greifer 1 muss verbunden sein, um dieses Programm auszuführen.", "Keine Verbindung", False, True, True)
      end
      if not(rq_is_gripper_activated("1")):
        popup("Greifer 1 ist nicht aktiviert. Wechseln Sie zur Registerkarte Installation > Greifer, um ihn zu aktivieren und das Programm erneut auszuführen.", "Nicht aktiviert", False, True, True)
      end
      rq_set_pos_spd_for(0, 255, 255, "1")
      rq_wait_pos_spe_for_request(0, 255, 255, "1")
      rq_go_to("1")
      rq_wait("1")
      # end: URCap Program Node
      $ 997 "FahreLinear"
      $ 998 "stn14_pk_rk_p" "breakAfter"
      set_tcp(p[-3.0E-4,2.5E-4,0.1575,0.0,0.0,0.0])
      movel(pose_trans(stn6_plane, pose_trans(p[.776557109756, -.878329076792, .250244777977, -.001605684562, .009314448336, 1.565629725105], stn14_pk_rk_p_p)), a=1.2, v=0.25)
      # begin: URCap Program Node
      #   Source: Robotiq_Grippers, 1.8.13.22852, Robotiq Inc.
      #   Type: Greifer
      $ 999 "Greifer geschlossen (1)"
      if not(gripper_connected[0]):
        popup("Greifer 1 muss verbunden sein, um dieses Programm auszuführen.", "Keine Verbindung", False, True, True)
      end
      if not(rq_is_gripper_activated("1")):
        popup("Greifer 1 ist nicht aktiviert. Wechseln Sie zur Registerkarte Installation > Greifer, um ihn zu aktivieren und das Programm erneut auszuführen.", "Nicht aktiviert", False, True, True)
      end
      rq_set_pos_spd_for(255, 64, 255, "1")
      rq_wait_pos_spe_for_request(255, 64, 255, "1")
      rq_go_to("1")
      rq_wait("1")
      # end: URCap Program Node
      $ 1000 "stn14_pkrk_up_p" "breakAfter"
      set_tcp(p[-3.0E-4,2.5E-4,0.1575,0.0,0.0,0.0])
      movel(pose_trans(stn6_plane, pose_trans(p[.776557109756, -.878329076792, .250244777977, -.001605684562, .009314448336, 1.565629725105], stn14_pkrk_up_p_p)), a=1.2, v=0.25)
      $ 1001 "FahreLinear"
      $ 1002 "stn14_stn8_hl_p" "breakAfter"
      set_tcp(p[-3.0E-4,2.5E-4,0.1575,0.0,0.0,0.0])
      movel(pose_trans(stn6_plane, pose_trans(p[.776557109756, -.878329076792, .250244777977, -.001605684562, .009314448336, 1.565629725105], stn14_stn8_hl_p_p)), a=1.0, v=0.2)
      $ 1003 "stn8_hlp_2_p" "breakAfter"
      set_tcp(p[-3.0E-4,2.5E-4,0.1575,0.0,0.0,0.0])
      movel(pose_trans(stn6_plane, pose_trans(p[.776557109756, -.878329076792, .250244777977, -.001605684562, .009314448336, 1.565629725105], stn8_hlp_2_p_p)), a=1.0, v=0.2)
      $ 1004 "stn8_home_p" "breakAfter"
      set_tcp(p[-3.0E-4,2.5E-4,0.1575,0.0,0.0,0.0])
      movel(pose_trans(stn6_plane, pose_trans(p[.776557109756, -.878329076792, .250244777977, -.001605684562, .009314448336, 1.565629725105], stn8_home_p_p)), a=1.0, v=0.2, r=0.1)
      $ 1005 "stn8_pl_apr1_p" "breakAfter"
      set_tcp(p[-3.0E-4,2.5E-4,0.1575,0.0,0.0,0.0])
      movel(pose_trans(stn6_plane, pose_trans(p[.776557109756, -.878329076792, .250244777977, -.001605684562, .009314448336, 1.565629725105], stn8_pl_apr1_p_p)), a=1.0, v=0.2)
      $ 1006 "stn8_pl_apr2_p" "breakAfter"
      set_tcp(p[-3.0E-4,2.5E-4,0.1575,0.0,0.0,0.0])
      movel(pose_trans(stn6_plane, pose_trans(p[.776557109756, -.878329076792, .250244777977, -.001605684562, .009314448336, 1.565629725105], stn8_pl_apr2_p_p)), a=0.5, v=0.05)
      $ 1007 "stn8_place_p" "breakAfter"
      set_tcp(p[-3.0E-4,2.5E-4,0.1575,0.0,0.0,0.0])
      movel(pose_trans(stn6_plane, pose_trans(p[.776557109756, -.878329076792, .250244777977, -.001605684562, .009314448336, 1.565629725105], stn8_place_p_p)), a=0.5, v=0.05)
      # begin: URCap Program Node
      #   Source: Robotiq_Grippers, 1.8.13.22852, Robotiq Inc.
      #   Type: Greifer
      $ 1008 "Greiferbewegung40% (1)"
      if not(gripper_connected[0]):
        popup("Greifer 1 muss verbunden sein, um dieses Programm auszuführen.", "Keine Verbindung", False, True, True)
      end
      if not(rq_is_gripper_activated("1")):
        popup("Greifer 1 ist nicht aktiviert. Wechseln Sie zur Registerkarte Installation > Greifer, um ihn zu aktivieren und das Programm erneut auszuführen.", "Nicht aktiviert", False, True, True)
      end
      rq_set_pos_spd_for(102, 64, 255, "1")
      rq_wait_pos_spe_for_request(102, 64, 255, "1")
      rq_go_to("1")
      rq_wait("1")
      # end: URCap Program Node
      $ 1009 "stn8_pl_apr2_p" "breakAfter"
      set_tcp(p[-3.0E-4,2.5E-4,0.1575,0.0,0.0,0.0])
      movel(pose_trans(stn6_plane, pose_trans(p[.776557109756, -.878329076792, .250244777977, -.001605684562, .009314448336, 1.565629725105], stn8_pl_apr2_p_p)), a=1.0, v=0.2)
      $ 1010 "stn8_pl_apr1_p" "breakAfter"
      set_tcp(p[-3.0E-4,2.5E-4,0.1575,0.0,0.0,0.0])
      movel(pose_trans(stn6_plane, pose_trans(p[.776557109756, -.878329076792, .250244777977, -.001605684562, .009314448336, 1.565629725105], stn8_pl_apr1_p_p)), a=1.0, v=0.2)
      # begin: URCap Program Node
      #   Source: Robotiq_Grippers, 1.8.13.22852, Robotiq Inc.
      #   Type: Greifer
      $ 1011 "Greifer geschlossen (1)"
      if not(gripper_connected[0]):
        popup("Greifer 1 muss verbunden sein, um dieses Programm auszuführen.", "Keine Verbindung", False, True, True)
      end
      if not(rq_is_gripper_activated("1")):
        popup("Greifer 1 ist nicht aktiviert. Wechseln Sie zur Registerkarte Installation > Greifer, um ihn zu aktivieren und das Programm erneut auszuführen.", "Nicht aktiviert", False, True, True)
      end
      rq_set_pos_spd_for(255, 255, 255, "1")
      rq_wait_pos_spe_for_request(255, 255, 255, "1")
      rq_go_to("1")
      rq_wait("1")
      # end: URCap Program Node
      $ 1012 "FahreAchse"
      $ 1013 "stn8_home_p" "breakAfter"
      set_tcp(p[-3.0E-4,2.5E-4,0.1575,0.0,0.0,0.0])
      movej(get_inverse_kin(pose_trans(stn6_plane, pose_trans(p[.776557109756, -.878329076792, .250244777977, -.001605684562, .009314448336, 1.565629725105], stn8_home_p_p)), qnear=stn8_home_p_q), a=1.3962634015954636, v=1.0471975511965976, r=0.1)
      $ 1014 "stn8_stn6_hlp_p" "breakAfter"
      set_tcp(p[-3.0E-4,2.5E-4,0.1575,0.0,0.0,0.0])
      movej(get_inverse_kin(pose_trans(stn6_plane, pose_trans(p[.776557109756, -.878329076792, .250244777977, -.001605684562, .009314448336, 1.565629725105], stn8_stn6_hlp_p_p)), qnear=stn8_stn6_hlp_p_q), a=1.3962634015954636, v=1.0471975511965976, r=0.1)
      $ 1015 "stn6_home_p" "breakAfter"
      set_tcp(p[-3.0E-4,2.5E-4,0.1575,0.0,0.0,0.0])
      movej(get_inverse_kin(pose_trans(stn6_plane, pose_trans(p[.776557109756, -.878329076792, .250244777977, -.001605684562, .009314448336, 1.565629725105], stn6_home_p_p)), qnear=stn6_home_p_q), a=1.3962634015954636, v=1.0471975511965976)
      $ 1016 "Aufruf reset_jobs"
      reset_jobs()
    elif (151 == switch_1):
      $ 1017 "Case 151"
      $ 1018 "dest_jobID≔jobArr[1]"
      global dest_jobID=jobArr[1]
      $ 1019 "FahreAchse"
      $ 1020 "stn1_home_p" "breakAfter"
      set_tcp(p[-3.0E-4,2.5E-4,0.1575,0.0,0.0,0.0])
      movej(get_inverse_kin(pose_trans(stn1_plane, pose_trans(p[.053539610991, -.984987293150, -.024848236577, .000189536594, .000276418508, 3.136265531618], stn1_home_p_p)), qnear=stn1_home_p_q), a=1.3962634015954636, v=1.0471975511965976)
      $ 1021 "Switch dest_jobID"
      switch_2 = dest_jobID
      $ 1022 "Case 72"
      if (72 == switch_2):
        $ 1023 "src_dest_p≔qMast.get_loc()"
        global src_dest_p=qMast.get_loc()
        $ 1024 "source_p≔src_dest_p[0]"
        global source_p=src_dest_p[0]
        $ 1025 "dest_p≔src_dest_p[1]"
        global dest_p=src_dest_p[1]
        $ 1026 "FahreAchse"
        $ 1027 "stn15_home_p" "breakAfter"
        set_tcp(p[-3.0E-4,2.5E-4,0.1575,0.0,0.0,0.0])
        movej(get_inverse_kin(pose_trans(stn6_plane, pose_trans(p[.776557109756, -.878329076792, .250244777977, -.001605684562, .009314448336, 1.565629725105], stn15_home_p_p)), qnear=stn15_home_p_q), a=1.3962634015954636, v=1.0471975511965976)
        $ 1028 "FahreLinear"
        $ 1029 "source_p" "breakAfter"
        set_tcp(p[-3.0E-4,2.5E-4,0.1575,0.0,0.0,0.0])
        movel(pose_trans(stn6_plane, source_p), a=1.2, v=0.25)
        # begin: URCap Program Node
        #   Source: Robotiq_Grippers, 1.8.13.22852, Robotiq Inc.
        #   Type: Greifer
        $ 1030 "Greiferbewegung50% (1)"
        if not(gripper_connected[0]):
          popup("Greifer 1 muss verbunden sein, um dieses Programm auszuführen.", "Keine Verbindung", False, True, True)
        end
        if not(rq_is_gripper_activated("1")):
          popup("Greifer 1 ist nicht aktiviert. Wechseln Sie zur Registerkarte Installation > Greifer, um ihn zu aktivieren und das Programm erneut auszuführen.", "Nicht aktiviert", False, True, True)
        end
        rq_set_pos_spd_for(128, 255, 255, "1")
        rq_wait_pos_spe_for_request(128, 255, 255, "1")
        rq_go_to("1")
        rq_wait("1")
        # end: URCap Program Node
        $ 1031 "cur_pose≔pose_trans(pose_inv(stn6_plane), get_actual_tcp_pose())"
        global cur_pose= pose_trans ( pose_inv (stn6_plane),  get_actual_tcp_pose ())
        $ 1032 "stn15_pk_z_p≔pose_trans(cur_pose, p[0,0,stn15_pick_z/1000,0,0,0])"
        global stn15_pk_z_p= pose_trans (cur_pose, p[0,0,stn15_pick_z/1000,0,0,0])
        $ 1033 "stn15_pk_z_p" "breakAfter"
        set_tcp(p[-3.0E-4,2.5E-4,0.1575,0.0,0.0,0.0])
        movel(pose_trans(stn6_plane, stn15_pk_z_p), a=0.5, v=0.1)
        # begin: URCap Program Node
        #   Source: Robotiq_Grippers, 1.8.13.22852, Robotiq Inc.
        #   Type: Greifer
        $ 1034 "Greifer geschlossen (1)"
        if not(gripper_connected[0]):
          popup("Greifer 1 muss verbunden sein, um dieses Programm auszuführen.", "Keine Verbindung", False, True, True)
        end
        if not(rq_is_gripper_activated("1")):
          popup("Greifer 1 ist nicht aktiviert. Wechseln Sie zur Registerkarte Installation > Greifer, um ihn zu aktivieren und das Programm erneut auszuführen.", "Nicht aktiviert", False, True, True)
        end
        rq_set_pos_spd_for(255, 128, 128, "1")
        rq_wait_pos_spe_for_request(255, 128, 128, "1")
        rq_go_to("1")
        rq_wait("1")
        # end: URCap Program Node
        $ 1035 "source_p" "breakAfter"
        set_tcp(p[-3.0E-4,2.5E-4,0.1575,0.0,0.0,0.0])
        movel(pose_trans(stn6_plane, source_p), a=1.2, v=0.25)
        $ 1036 "stn15_home_p" "breakAfter"
        set_tcp(p[-3.0E-4,2.5E-4,0.1575,0.0,0.0,0.0])
        movel(pose_trans(stn6_plane, pose_trans(p[.776557109756, -.878329076792, .250244777977, -.001605684562, .009314448336, 1.565629725105], stn15_home_p_p)), a=1.2, v=0.25)
        $ 1037 "FahreAchse"
        $ 1038 "stn7_home_p" "breakAfter"
        set_tcp(p[-3.0E-4,2.5E-4,0.1575,0.0,0.0,0.0])
        movej(get_inverse_kin(pose_trans(stn7_plane, pose_trans(p[.109811488584, -1.023382701287, -.166619380160, .003048702642, -.008599620441, 2.442192581404], stn7_home_p_p)), qnear=stn7_home_p_q), a=1.3962634015954636, v=1.0471975511965976, r=0.1)
        $ 1039 "Aufruf stn7_check_doors"
        stn7_check_doors()
        $ 1040 "FahreLinear"
        $ 1041 "dest_p" "breakAfter"
        set_tcp(p[-3.0E-4,2.5E-4,0.1575,0.0,0.0,0.0])
        movel(pose_trans(stn7_plane, dest_p), a=1.2, v=0.25)
        $ 1042 "cur_pose≔pose_trans(pose_inv(stn7_plane), get_actual_tcp_pose())"
        global cur_pose= pose_trans ( pose_inv (stn7_plane),  get_actual_tcp_pose ())
        $ 1043 "stn7_place_p≔pose_trans(cur_pose, p[0,0,stn7_place_z/1000,0,0,0])"
        global stn7_place_p= pose_trans (cur_pose, p[0,0,stn7_place_z/1000,0,0,0])
        $ 1044 "FahreLinear"
        $ 1045 "stn7_place_p" "breakAfter"
        set_tcp(p[-3.0E-4,2.5E-4,0.1575,0.0,0.0,0.0])
        movel(pose_trans(stn7_plane, stn7_place_p), a=0.15, v=0.075)
        # begin: URCap Program Node
        #   Source: Robotiq_Grippers, 1.8.13.22852, Robotiq Inc.
        #   Type: Greifer
        $ 1046 "Greifer offen (1)"
        if not(gripper_connected[0]):
          popup("Greifer 1 muss verbunden sein, um dieses Programm auszuführen.", "Keine Verbindung", False, True, True)
        end
        if not(rq_is_gripper_activated("1")):
          popup("Greifer 1 ist nicht aktiviert. Wechseln Sie zur Registerkarte Installation > Greifer, um ihn zu aktivieren und das Programm erneut auszuführen.", "Nicht aktiviert", False, True, True)
        end
        rq_set_pos_spd_for(0, 255, 255, "1")
        rq_wait_pos_spe_for_request(0, 255, 255, "1")
        rq_go_to("1")
        rq_wait("1")
        # end: URCap Program Node
        $ 1047 "FahreLinear"
        $ 1048 "dest_p" "breakAfter"
        set_tcp(p[-3.0E-4,2.5E-4,0.1575,0.0,0.0,0.0])
        movel(pose_trans(stn7_plane, dest_p), a=1.2, v=0.25)
        # begin: URCap Program Node
        #   Source: Robotiq_Grippers, 1.8.13.22852, Robotiq Inc.
        #   Type: Greifer
        $ 1049 "Greifer geschlossen (1)"
        if not(gripper_connected[0]):
          popup("Greifer 1 muss verbunden sein, um dieses Programm auszuführen.", "Keine Verbindung", False, True, True)
        end
        if not(rq_is_gripper_activated("1")):
          popup("Greifer 1 ist nicht aktiviert. Wechseln Sie zur Registerkarte Installation > Greifer, um ihn zu aktivieren und das Programm erneut auszuführen.", "Nicht aktiviert", False, True, True)
        end
        rq_set_pos_spd_for(255, 255, 255, "1")
        rq_wait_pos_spe_for_request(255, 255, 255, "1")
        rq_go_to("1")
        rq_wait("1")
        # end: URCap Program Node
        $ 1050 "FahreAchse"
        $ 1051 "stn7_home_p" "breakAfter"
        set_tcp(p[-3.0E-4,2.5E-4,0.1575,0.0,0.0,0.0])
        movej(get_inverse_kin(pose_trans(stn7_plane, pose_trans(p[.109811488584, -1.023382701287, -.166619380160, .003048702642, -.008599620441, 2.442192581404], stn7_home_p_p)), qnear=stn7_home_p_q), a=1.3962634015954636, v=1.0471975511965976)
        $ 1052 "Aufruf reset_jobs"
        reset_jobs()
      end
    end
  end
end
